// TIA Portal V17 export
// export: Created 2024-08-09T12:53:21.8743715Z, ExportSetting WithDefaults, DisplayName Totally Integrated Automation Portal, DisplayVersion V17 Update 7, DisplayName TIA Portal Openness, DisplayVersion V17 Update 7, DisplayName TIA Portal Version Control Interface, DisplayVersion V17, DisplayName STEP 7 Professional, DisplayVersion V17 Update 7, DisplayName STEP 7 Safety, DisplayVersion V17 Update 6, DisplayName WinCC Professional, DisplayVersion V17 Update 7
TYPE "S_ChargPont"
// stored: IsFailsafeCompliant false
   STRUCT
      _Ptzs : "S_SuiviCommande";
      _Commande { S7_SetPoint := 'True'} : "S_ComLign";
      _Circuit { ExternalAccessible := 'False'; ExternalVisible := 'False'; ExternalWritable := 'False'} : "S_Circuit";
      _ChargCommun : "S_ChargCommun";
      _VidCel { S7_SetPoint := 'True'} : "VidCel";
      _TabMobIncomp { ExternalAccessible := 'False'; ExternalVisible := 'False'; ExternalWritable := 'False'} : Array[0.."MAX_MOB_INCOMP"] of "S_MobIncomp";
      Dial_Def { ExternalAccessible := 'False'; ExternalVisible := 'False'; ExternalWritable := 'False'} : "S_DIALOG_DEF";
      _ListeTaAttAutDemarrage { ExternalAccessible := 'False'; ExternalVisible := 'False'; ExternalWritable := 'False'} : Array[0.."T_MAX_AMONTAVAL"] of "S_TacheNiv";
      _ListeTaAttCtrlColChute { ExternalAccessible := 'False'; ExternalVisible := 'False'; ExternalWritable := 'False'} : Array[0.."T_MAX_AMONTAVAL"] of "S_TacheNiv";
      _ListeTaAttFinVidCompo { ExternalAccessible := 'False'; ExternalVisible := 'False'; ExternalWritable := 'False'} : Array[0.."T_MAX_AMONTAVAL"] of "S_TacheNiv";
      _ListeTaPositCamionOK { ExternalAccessible := 'False'; ExternalVisible := 'False'; ExternalWritable := 'False'} : Array[0.."T_MAX_AMONTAVAL"] of "S_TacheNiv";
      _ListeTaAttFinCharg { ExternalAccessible := 'False'; ExternalVisible := 'False'; ExternalWritable := 'False'} : Array[0.."T_MAX_AMONTAVAL"] of "S_TacheNiv";
      CycleOF { ExternalAccessible := 'False'; ExternalVisible := 'False'; ExternalWritable := 'False'} : Struct   // cycle ouverture fermeture ext
         _DebOuv { ExternalAccessible := 'False'; ExternalVisible := 'False'; ExternalWritable := 'False'} : Date_And_Time;
         _TpsPicke { ExternalAccessible := 'False'; ExternalVisible := 'False'; ExternalWritable := 'False'} : Date_And_Time;
         _Debut { ExternalAccessible := 'False'; ExternalVisible := 'False'; ExternalWritable := 'False'} : Date_And_Time;
         _TpsOuv { ExternalAccessible := 'False'; ExternalVisible := 'False'; ExternalWritable := 'False'} : Time;
         _TpCycleOuv { ExternalAccessible := 'False'; ExternalVisible := 'False'; ExternalWritable := 'False'} : Time;
         _PoidsPrec { ExternalAccessible := 'False'; ExternalVisible := 'False'; ExternalWritable := 'False'} : Real;
         _FgDef { ExternalAccessible := 'False'; ExternalVisible := 'False'; ExternalWritable := 'False'} : Bool;
      END_STRUCT;
      CtrlEvol { ExternalAccessible := 'False'; ExternalVisible := 'False'; ExternalWritable := 'False'} : Struct   // cycle ouverture fermeture ext
         _TpsRestant { ExternalAccessible := 'False'; ExternalVisible := 'False'; ExternalWritable := 'False'} : Date_And_Time;
         _TpsPicke { ExternalAccessible := 'False'; ExternalVisible := 'False'; ExternalWritable := 'False'} : Date_And_Time;
         _Debut { ExternalAccessible := 'False'; ExternalVisible := 'False'; ExternalWritable := 'False'} : Date_And_Time;
         _PoidsPrec { ExternalAccessible := 'False'; ExternalVisible := 'False'; ExternalWritable := 'False'} : Real;
         _FgDef { ExternalAccessible := 'False'; ExternalVisible := 'False'; ExternalWritable := 'False'} : Bool;
      END_STRUCT;
      CalcDebit : Struct   // Calcul debit du pont
         _TpsPicke { ExternalAccessible := 'False'; ExternalVisible := 'False'; ExternalWritable := 'False'} : Date_And_Time;
         _TpCalcDebit { ExternalAccessible := 'False'; ExternalVisible := 'False'; ExternalWritable := 'False'} : Time;   // Tempo calcul debit pont de chargement
         _TabPoids { ExternalAccessible := 'False'; ExternalVisible := 'False'; ExternalWritable := 'False'} : Array[0..11] of Real;
         _DebitPont : Real;   // Debit pont
         _Ecart { ExternalAccessible := 'False'; ExternalVisible := 'False'; ExternalWritable := 'False'} : Real;
         _NbPoidsCalcDebit { ExternalAccessible := 'False'; ExternalVisible := 'False'; ExternalWritable := 'False'} : Int;   // Nombre de poids memorise pour calculer le debit
         _PremFois { ExternalAccessible := 'False'; ExternalVisible := 'False'; ExternalWritable := 'False'} : Bool;
      END_STRUCT;
      _TpsPicke { ExternalAccessible := 'False'; ExternalVisible := 'False'; ExternalWritable := 'False'} : Date_And_Time;
      _DebStable { ExternalAccessible := 'False'; ExternalVisible := 'False'; ExternalWritable := 'False'} : Date_And_Time;
      _DebFermExt { ExternalAccessible := 'False'; ExternalVisible := 'False'; ExternalWritable := 'False'} : Date_And_Time;
      _Debut { ExternalAccessible := 'False'; ExternalVisible := 'False'; ExternalWritable := 'False'} : Date_And_Time;
      _TpPoidsStab { ExternalAccessible := 'False'; ExternalVisible := 'False'; ExternalWritable := 'False'} : Time;   // Temps pendant lequel le poids doit etre stable
      _TpCycleOuverture { ExternalAccessible := 'False'; ExternalVisible := 'False'; ExternalWritable := 'False'} : Time;   // Tempo d'ouverture de la trappe qui va permettre de calculer le nombre d'ouverture pour avoir la quantitÃ© voulue
      _TpCycleFermeture { ExternalAccessible := 'False'; ExternalVisible := 'False'; ExternalWritable := 'False'} : Time;   // Tempo de fermeture entre deux extractions
      _TpRestOuv { ExternalAccessible := 'False'; ExternalVisible := 'False'; ExternalWritable := 'False'} : Time;   // Tempo restant avant la fermeture du cycle d'extraction
      _PoidsCycle { ExternalAccessible := 'False'; ExternalVisible := 'False'; ExternalWritable := 'False'} : Real;
      _PoidsPont { ExternalAccessible := 'False'; ExternalVisible := 'False'; ExternalWritable := 'False'} : Real;
      _PoidsPrec { ExternalAccessible := 'False'; ExternalVisible := 'False'; ExternalWritable := 'False'} : Real;
      _MinChute { ExternalAccessible := 'False'; ExternalVisible := 'False'; ExternalWritable := 'False'} : Real;   // Colonne de chute minimum
      _MaxChute { ExternalAccessible := 'False'; ExternalVisible := 'False'; ExternalWritable := 'False'} : Real;   // Colonne de chute maximum
      _MaxChuteTamis { ExternalAccessible := 'False'; ExternalVisible := 'False'; ExternalWritable := 'False'} : Real;   // Colonne de chute maximum avec tamiseur
      _MaxCorChute { ExternalAccessible := 'False'; ExternalVisible := 'False'; ExternalWritable := 'False'} : Real;   // Correction maximum de la colonne de chute
      _EcartPoidsStab { ExternalAccessible := 'False'; ExternalVisible := 'False'; ExternalWritable := 'False'} : Real;   // Ecart maximum poids considerer le poids Stable
      _TolDernCase { ExternalAccessible := 'False'; ExternalVisible := 'False'; ExternalWritable := 'False'} : Real;
      _ConsArrCalcColChute { ExternalAccessible := 'False'; ExternalVisible := 'False'; ExternalWritable := 'False'} : Real;   // Consigne d'arret pour calcul colonne de chute
      _TolVideCel { ExternalAccessible := 'False'; ExternalVisible := 'False'; ExternalWritable := 'False'} : Real;   // Tolerance de quantite pendant une vide cellule
      _MemoPoids { ExternalAccessible := 'False'; ExternalVisible := 'False'; ExternalWritable := 'False'} : Real;
      _LectChute { ExternalAccessible := 'False'; ExternalVisible := 'False'; ExternalWritable := 'False'} : Int;   // Lecture colonne de chute en base
      _Fpv { ExternalAccessible := 'False'; ExternalVisible := 'False'; ExternalWritable := 'False'} : Int;
      _ChuteArrImm { ExternalAccessible := 'False'; ExternalVisible := 'False'; ExternalWritable := 'False'} : Int;   // Colonne de chute applique sur un arret immediat
      _TolEcTare { ExternalAccessible := 'False'; ExternalVisible := 'False'; ExternalWritable := 'False'} : Int;   // Ecart maximum possible entre la pese burt de la commande prec et la tare de la commande EC
      _ExtCons { ExternalAccessible := 'False'; ExternalVisible := 'False'; ExternalWritable := 'False'} : Int;   // Consigne d'extractions
      _MbTamis { ExternalAccessible := 'False'; ExternalVisible := 'False'; ExternalWritable := 'False'} : Int := -1;   // Mobile tamiseur
      _MobInc { ExternalAccessible := 'False'; ExternalVisible := 'False'; ExternalWritable := 'False'} : Int;
      _ExtReel { ExternalAccessible := 'False'; ExternalVisible := 'False'; ExternalWritable := 'False'} : USInt;   // Nombre d'extractions realisees
      _IndexTemp { ExternalAccessible := 'False'; ExternalVisible := 'False'; ExternalWritable := 'False'} : USInt;
      _NbRelAutoExp { ExternalAccessible := 'False'; ExternalVisible := 'False'; ExternalWritable := 'False'} : USInt;   // Nombre de relance automatique du chargement
      _FgTypeLancColChute { ExternalAccessible := 'False'; ExternalVisible := 'False'; ExternalWritable := 'False'} : USInt;   // Type de lancement lorsque la colonne de chute est superieure a la consigne (0: debit, 1: bouton Ajout, 2: cycle d'ouverture de la trappe)
      _NbRelAuto { ExternalAccessible := 'False'; ExternalVisible := 'False'; ExternalWritable := 'False'} : USInt;
      _MemoVit { ExternalAccessible := 'False'; ExternalVisible := 'False'; ExternalWritable := 'False'} : USInt;
      _Bouton { ExternalAccessible := 'False'; ExternalVisible := 'False'; ExternalWritable := 'False'} : USInt;
      _FgCycleOuverture { ExternalAccessible := 'False'; ExternalVisible := 'False'; ExternalWritable := 'False'} : USInt;   // Flag indiquant que l'ouverture est terminee
      _BtDemTare : USInt;   // Bouton supervision demande Tare
      _BtDepCycle : USInt;   // Bouton supervision depart cycle
      _BtAdandonLigne : USInt;   // Bouton supervision abndon ligne de chargement
      _BtSusp : USInt;   // Bouton supervision Suspension chargement
      _BtAjout : USInt;   // Bouton supervision Ajout produit
      _BtChgCellule : USInt;   // Bouton supervision changement cellule
      _MemoAppuiBP { ExternalAccessible := 'False'; ExternalVisible := 'False'; ExternalWritable := 'False'} : USInt;
      _DemChgtCase { ExternalAccessible := 'False'; ExternalVisible := 'False'; ExternalWritable := 'False'} : USInt;   // Flag de demande de changement de case
      _MemoEtapeBt { ExternalAccessible := 'False'; ExternalVisible := 'False'; ExternalWritable := 'False'} : SInt;   // memorisation etape pour gestion de bouton
      _NbRelDefArrProd { ExternalAccessible := 'False'; ExternalVisible := 'False'; ExternalWritable := 'False'} : SInt;
      _MemoRajout { ExternalAccessible := 'False'; ExternalVisible := 'False'; ExternalWritable := 'False'} : Bool;
      _ValidPasArriveeProduit { ExternalAccessible := 'False'; ExternalVisible := 'False'; ExternalWritable := 'False'} : Bool;   // Validation controle arrivee produit
      _BpDemTare { ExternalAccessible := 'False'; ExternalVisible := 'False'; ExternalWritable := 'False'} : Bool;   // Bouton poussoir demande Tare
      _BpDepCycle { ExternalAccessible := 'False'; ExternalVisible := 'False'; ExternalWritable := 'False'} : Bool;   // Bouton poussoir depart cycle
      _BpSusp { ExternalAccessible := 'False'; ExternalVisible := 'False'; ExternalWritable := 'False'} : Bool;   // Bouton poussoir suspension chargement
      _BpAjout { ExternalAccessible := 'False'; ExternalVisible := 'False'; ExternalWritable := 'False'} : Bool;   // Bouton poussoir ajout produit
      _FgEtiqDebutChar { ExternalAccessible := 'False'; ExternalVisible := 'False'; ExternalWritable := 'False'} : Bool;   // validation impreesion etiquette en debut de chargement
      _PriseTareAvDem { ExternalAccessible := 'False'; ExternalVisible := 'False'; ExternalWritable := 'False'} : Bool;   // Attente Prise tare avant demarrage
      _DefLiaison { ExternalAccessible := 'False'; ExternalVisible := 'False'; ExternalWritable := 'False'} : Bool;   // Defaut liaison benne peseuse
      _HorsGamme { ExternalAccessible := 'False'; ExternalVisible := 'False'; ExternalWritable := 'False'} : Bool;   // Flag hors Gamme
      _ChargDebit { ExternalAccessible := 'False'; ExternalVisible := 'False'; ExternalWritable := 'False'} : Bool;   // Chargement sur Debit
      _ChargCycle { ExternalAccessible := 'False'; ExternalVisible := 'False'; ExternalWritable := 'False'} : Bool;   // Chargement sur cycle d'ouverture
      _AttRelBt { ExternalAccessible := 'False'; ExternalVisible := 'False'; ExternalWritable := 'False'} : Bool;   // Attente relance bouton
      _FgParamAuto { ExternalAccessible := 'False'; ExternalVisible := 'False'; ExternalWritable := 'False'} : Bool;   // Parametre automatisme existant pour l'expedition
      _ConfFinDefEvol { ExternalAccessible := 'False'; ExternalVisible := 'False'; ExternalWritable := 'False'} : Bool;   // confirmation de fin de chargement en cas de defaut evolution + tolerance
      _CtrlPoidsHorsPont { ExternalAccessible := 'False'; ExternalVisible := 'False'; ExternalWritable := 'False'} : Bool;   // Controle poids du pont en mode HORS PONT
      _VidAuto { ExternalAccessible := 'False'; ExternalVisible := 'False'; ExternalWritable := 'False'} : Bool;   // Vidange automatique lorsque la quantie a atteint la consigne
      _ChargTelem { ExternalAccessible := 'False'; ExternalVisible := 'False'; ExternalWritable := 'False'} : Bool;   // Parametre pour savoir si c'est un chargement avec telemetre
      _AutorMAJColChute { ExternalAccessible := 'False'; ExternalVisible := 'False'; ExternalWritable := 'False'} : Bool;
      _ArrImmMemeProd { ExternalAccessible := 'False'; ExternalVisible := 'False'; ExternalWritable := 'False'} : Bool;   // Possibilite Arret immediat circuit si circuit identique
      _SuspCircuit { ExternalAccessible := 'False'; ExternalVisible := 'False'; ExternalWritable := 'False'} : Bool;   // Flag de suspension chargement
      _ChgtCelAuto { ExternalAccessible := 'False'; ExternalVisible := 'False'; ExternalWritable := 'False'} : Bool;   // Changement cellule automatique
      _ParamTrouve { ExternalAccessible := 'False'; ExternalVisible := 'False'; ExternalWritable := 'False'} : Bool;
      _ActionAvantDemarCircuit { ExternalAccessible := 'False'; ExternalVisible := 'False'; ExternalWritable := 'False'} : Bool;
      _ActionApresDemarCircuit { ExternalAccessible := 'False'; ExternalVisible := 'False'; ExternalWritable := 'False'} : Bool;
      _ActionAvantVidangeCircuit { ExternalAccessible := 'False'; ExternalVisible := 'False'; ExternalWritable := 'False'} : Bool;
      _ActionApresVidangeCircuit { ExternalAccessible := 'False'; ExternalVisible := 'False'; ExternalWritable := 'False'} : Bool;
      _ActionApresArretImm { ExternalAccessible := 'False'; ExternalVisible := 'False'; ExternalWritable := 'False'} : Bool;
      _ActionPendantChargement { ExternalAccessible := 'False'; ExternalVisible := 'False'; ExternalWritable := 'False'} : Bool;
      _MemoDemChgCel { ExternalAccessible := 'False'; ExternalVisible := 'False'; ExternalWritable := 'False'} : Bool;
      _GestQteCaseAuto { ExternalAccessible := 'False'; ExternalVisible := 'False'; ExternalWritable := 'False'} : Bool;   // Gestion des quantite case
      _DemVib { ExternalAccessible := 'False'; ExternalVisible := 'False'; ExternalWritable := 'False'} : Bool;
   END_STRUCT;
END_TYPE
